Staubli VAL3: type1.pjx

--- type1.pjx ---
Parameters version=s7.6.2 stackSize=5000 millimeterUnit=true
Data file=type1.dtx
Type name=TrajSmallBox path=Disk://goHome/template/TrajSmallBox/TrajSmallBox.pjx

--- type1.dtx ---
public TrajSmallBox box{}
